TYPE ST_Event :
STRUCT
	eEventType: E_EventType; 
	eEventSeverity: TcEventSeverity;
	nEventIdentity: UDINT;
	sEventText: STRING(255);
	dtTimestamp: DATE_AND_TIME;
	
END_STRUCT
END_TYPE

(* stored: Version 1.1.0.1, ProductVersion 3.1.4024.12
   DUT ST_Event: Id {ca8b0247-8ca1-4b22-88d3-1e68121912c6} *)
